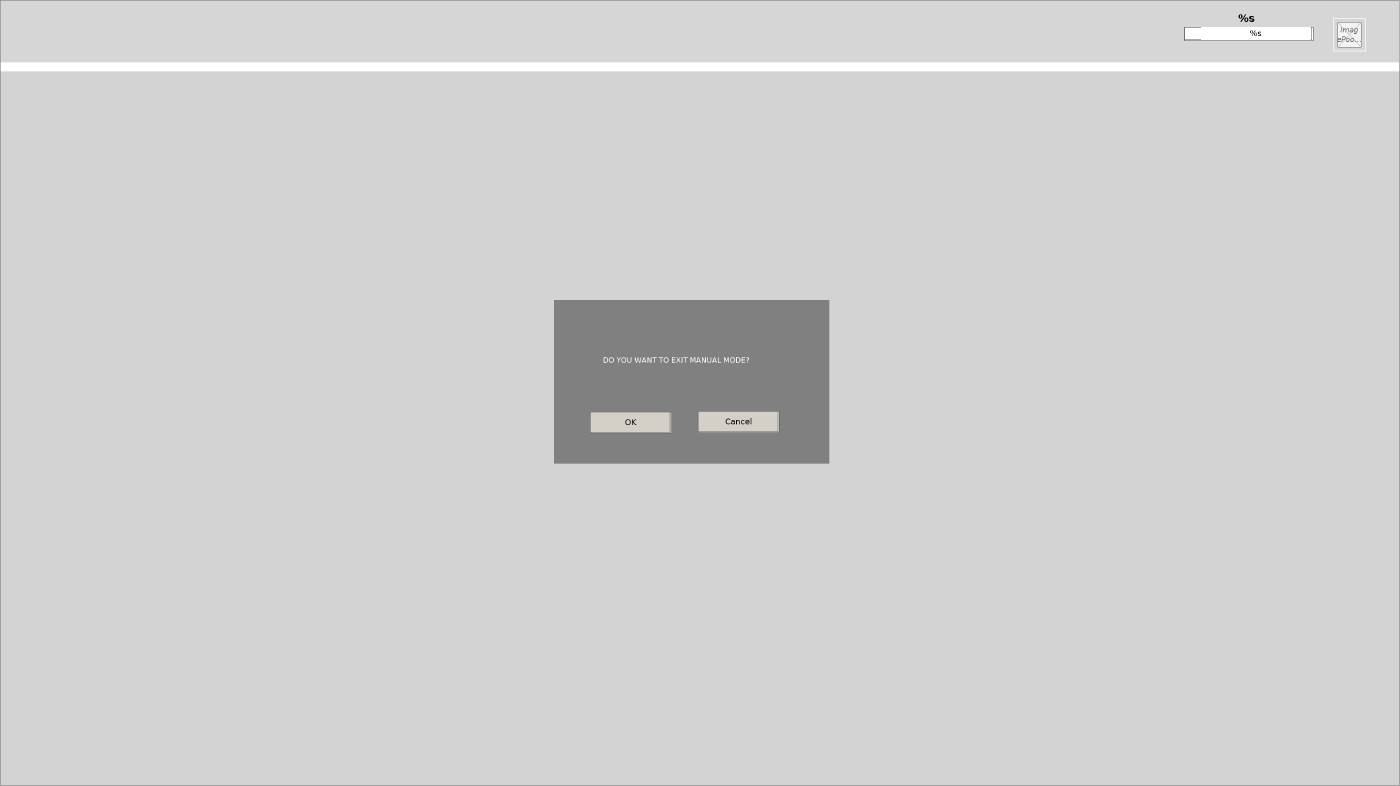
VISUALIZATION Manual_Exit_Popup  // 1920x1079
    Rectangle (0,98 1920x981)
    Rectangle (0,63 1920x26)
        p3528305787: HMI_Ctrl.ANIMATION3
    Rectangle (0,0 1919x85)
    Group (1828,25 45x45)
        OnMouseClick: toggle HMI_Ctrl.MenuButton
        RoundedRectangle (0,0 45x45), colour toggle: HMI_Ctrl.MenuButton
        Image (6,5 33x35), image: ImagePool.Menu Button
    Rectangle (760,412 377x224)
    Label (809,413 209x24)
    Label (824,469 241x51), "DO YOU WANT TO EXIT MANUAL MODE?"
    Button (809,565 112x30), "OK"
        tap bManualExitConfirm
    Button (957,564 112x30), "Cancel"
        tap bManualExitCancel
    Group (1621,14 180x42)
        Rectangle (0,0 177x22), "%s", text variable: DSLocalSystemTimeML.sCurrentDT24Hr_General
        Button (3,23 177x19), image: VisuSymbols.Symbols.AddUser
        Rectangle (26,23 150x18), "%s", text variable: fbHmiTF1800_UserlevelManagement.dsHmiUserStatus_Active.sLoginName
END_VISUALIZATION

(* stored: Version 1.1.0.1, ProductVersion 3.1.4024.12
   Visu Manual_Exit_Popup: Id {26e71f4b-ed93-4041-883d-38e771f97921} *)
